# EPICS substitutions: AutonomousMinimizationApp/Db/common/program.substitutions
file program.template
{
    {AREA="DIAG0",EXEC="EMIT", EXEC2 = "GPSR"}
}
